PROGRAM PosConfirmBitCtrl_Arm1
VAR

	fbFBPArmHorzZoneConfirm_Arm1 : fbV2_FBPArmHorzZoneConfirm;

END_VAR

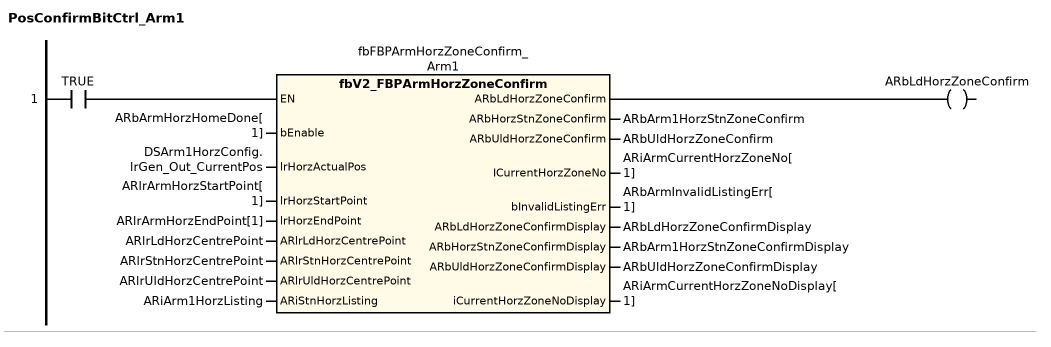
// NETWORK 1
fbFBPArmHorzZoneConfirm_Arm1(
    bEnable := ARbArmHorzHomeDone[1],
    lrHorzActualPos := DSArm1HorzConfig.lrGen_Out_CurrentPos,
    lrHorzStartPoint := ARlrArmHorzStartPoint[1],
    lrHorzEndPoint := ARlrArmHorzEndPoint[1],
    ARlrLdHorzCentrePoint := ARlrLdHorzCentrePoint,
    ARlrStnHorzCentrePoint := ARlrStnHorzCentrePoint,
    ARlrUldHorzCentrePoint := ARlrUldHorzCentrePoint,
    ARiStnHorzListing := ARiArm1HorzListing,
    ARbHorzStnZoneConfirm => ARbArm1HorzStnZoneConfirm,
    ARbUldHorzZoneConfirm => ARbUldHorzZoneConfirm,
    ICurrentHorzZoneNo => ARiArmCurrentHorzZoneNo[1],
    bInvalidListingErr => ARbArmInvalidListingErr[1],
    ARbLdHorzZoneConfirmDisplay => ARbLdHorzZoneConfirmDisplay,
    ARbHorzStnZoneConfirmDisplay => ARbArm1HorzStnZoneConfirmDisplay,
    ARbUldHorzZoneConfirmDisplay => ARbUldHorzZoneConfirmDisplay,
    iCurrentHorzZoneNoDisplay => ARiArmCurrentHorzZoneNoDisplay[1]); // fbV2_FBPArmHorzZoneConfirm
ARbLdHorzZoneConfirm := fbFBPArmHorzZoneConfirm_Arm1.ARbLdHorzZoneConfirm;

END_PROGRAM

(* stored: Version 1.1.0.1, ProductVersion 3.1.4024.12
   POU PosConfirmBitCtrl_Arm1: Id {3dcea65b-c342-4bff-b1df-821553f095cd}, SpecialFunc None *)
